TYPE "Peeler_Manager"
VERSION : 0.1
// Block: Peeler_Manager
   STRUCT
      Lift : ValveMachine_Manager;
      Extension : ValveMachine_Manager;
      FreeMovementAllowed : Bool;
      Move_Up_DecoilerChange : Bool;
      Move_Dwn_MaterialFeed : Bool;
   END_STRUCT;

END_TYPE
